{attribute 'GeneratedUsingTerminal: EP9521-0020-0000'}
{attribute addProperty BoxType "EP9521-0020-0000"}
{attribute addProperty Id "A_0025_EP9576_1032_0016EP9576_C42142C629"}
{attribute addProperty CRC "485439160"}
{attribute addProperty Size "29"}
TYPE A_0024_EP9521_0020_0000_1CEF36B8 EXTENDS EP9521_1FC0878B :
STRUCT
	{attribute addProperty Name "A_0025_EP9576_1032_0016"}
	{attribute addProperty PreviousPort "A_0024(EP9521-0020-0000) : B"}
	A_0025_EP9576_1032_0016 : EP9576_C42142C6;
END_STRUCT
END_TYPE

(* stored: Version 1.2.0.0, ProductVersion 3.1.4024.9
   DUT A_0024_EP9521_0020_0000_1CEF36B8: Id {d94ec863-caac-4251-b49a-311311b3587f} *)
